FUNCTION_BLOCK TIMER_SET_S (* Sets output for a timer in seconds *)
  (* Standard: 61499-2 *)
  (* Version 1.0, 09-01-12, Guilherme Jarentchuk, Universidade do Estado de Santa Catarina *)
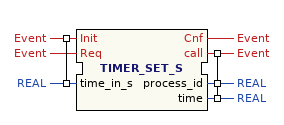
  EVENT_INPUT
    Init WITH time_in_s; (* Initialize execution *)
    Req; (* Request to finish *)
  END_EVENT
  EVENT_OUTPUT
    Cnf; (* Confirm execution *)
    call WITH process_id, time; (* Call execution device *)
  END_EVENT
  VAR_INPUT
    time_in_s : REAL;
  END_VAR
  VAR_OUTPUT
    process_id : REAL;
    time : REAL;
  END_VAR
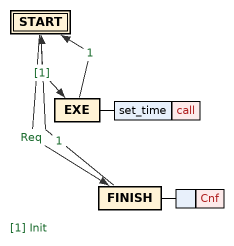
  EC_STATES
    START;
    EXE : set_time -> call;
    FINISH : -> Cnf;
  END_STATES
  EC_TRANSITIONS
    START TO EXE := Init;
    START TO FINISH := Req;
    EXE TO START := 1;
    FINISH TO START := 1;
  END_TRANSITIONS
  ALGORITHM set_time IN Lua:
time = time_in_s
process_id = -6
  END_ALGORITHM
END_FUNCTION_BLOCK
